(* CODESYS project HotWaterTank_student (2) (2).project

Project tree, tasks and I/O mapping:
  Device : CODESYS Control Win V3, 3S - Smart Software Solutions GmbH, version 3.5.17.10
    application Application
      libraries: Standard, * (System); Util, * (System)
      task MainTask (cyclic, interval t#10ms, priority 1) calls Model, PLC_PRG
      program Model [ST]: HeatingACT, SensorsACT, WaterLevelACT, OverpressureACT, InitializationACT
      visualisation Visualization
      program PLC_PRG [SFC]: Fill_active, Preheat_active_1, Operate_active, Init_Operate_active_active, Step0_Operate_active_active, Shutdown_active, HeatControl_active, Init_HeatControl_active_active, Step0_HeatControl_active_active, Empty_active, Fill_entry, Fill_exit, Preheat_entry, Preheat_exit, Operate_entry, Operate_exit, Shutdown_entry, Shutdown_exit, Empty_entry, Empty_exit
      trace Trace (task MainTask): Model.realTankLevel, Model.temperature
      global variables GVL
      function block GeneerinenSaato [ST]
      function block Heater [ST]
      function block SlowInlet [ST]
      function block FastInlet [ST]
      function block Heater2 [FBD]
      function block SlowInlet2 [FBD]
      function block FastInlet2 [FBD]
      visualisation Valvomo
  text list GlobalTextList
*)

// Device/Application/GVL
VAR_GLOBAL
	// Sensors:
	MinLevel:BOOL;
	LowLevel:BOOL;
	HighLevel:BOOL;
	MaxLevel:BOOL;
	MinTemp:BOOL;
	MaxTemp:BOOL;
	// Actuators:
	InletFast:BOOL;
	InletSlow:BOOL;
	Outlet:BOOL;
	Heat:BOOL;
END_VAR

// Device/Application/Model
PROGRAM Model
VAR
	// Define here the characteristics of the system.
	initialLevel :REAL := 0;		// Initial tank level, range [0..450], where 0=empty, 450=full tank.
	slowInlet :REAL := 10.0;		// Slow inlet flow rate in liters/s.
	fastInlet :REAL := 20.0;		// Fast inlet flow rate in liters/s.
	outlet	  :REAL := 15.0;		// Outlet flow rate in liters/s.
	posMinSensor	:REAL := 120;	// Position of min. sensor inside the tank. Range [0..450].
	posLowerSensor	:REAL := 170;	// Position of lower sensor inside the tank. Range [0..450].
	posUpperSensor	:REAL := 325;	// Position of upper sensor inside the tank. Range [0..450].
	posMaxSensor	:REAL := 375;	// Position of max sensor inside the tank. Range [0..450].
	minTemp   :REAL	:= 40.0;		// Minimum temperature sensor. Range [20..120].
	maxTemp   :REAL	:= 80.0;		// Maximum temperature sensor. Range [20..120].	
	heatCoeff :REAL := 3.0;			// Heating strenght of resistance.
	heatLooseCoeff	:REAL := 2.0;	// Cooling down coefficient of water.
END_VAR

VAR
	// Do not modify following variables unless you know what you are doing.
	initialized :BOOL := FALSE;
	tankLevel :REAL := 450.0;
	cycleTime :REAL := 10;			// PLC cycle time in ms. This should match the actual cycletime of the PLC.
	virtualTankLevel :REAL :=450;
	realTankLevel :REAL;
	slowValve :BOOL;
	fastValve :BOOL;
	outValve  :BOOL;
	heating   :BOOL;
	danger    :BOOL;
	overpress :REAL :=0.0;
	minSensor :BOOL;
	lowerSensor :BOOL;
	upperSensor :BOOL;
	maxSensor :BOOL;
	temperature :REAL :=20.0;
	minTempSensor :BOOL;
	maxTempSensor :BOOL;
	resistColor :DWORD := 16#00FF3A3A;
	resistBroken :BOOL;
	overheat :BOOL;
	tankExploded :BOOL;
	errorMsg :BOOL;
	blinkMsg :BLINK;
	startTrace :BOOL;
END_VAR

// Initialize system, only during reset.
IF NOT(initialized) THEN
	InitializationACT();
END_IF

// Read inputs from the controller's outputs:
IF NOT(tankExploded) THEN
	fastValve := GVL.InletFast;
	slowValve := GVL.InletSlow;
	outValve := GVL.Outlet;
	heating := GVL.Heat;
	startTrace := TRUE;
END_IF

// Determine the water level of tank based on inputs.
WaterLevelACT();

// Detect overpressure situations.
OverpressureACT();

// Run function taking care of the heating.
HeatingACT();

// Update sensors.
SensorsACT();

// Update model outputs / controller inputs:
GVL.MinLevel := minSensor;
GVL.LowLevel := lowerSensor;
GVL.HighLevel := upperSensor;
GVL.MaxLevel := maxSensor;
GVL.MinTemp := minTempSensor;
GVL.MaxTemp := maxTempSensor;

ACTION HeatingACT:
// Implementation of the heating
// Heating based on the level of the tank: the more water there is,
// the temperature will rise slower. Temperature refers to water temperature,
// not heating resistance.
IF heating AND (temperature < 100) AND (tankLevel < 449.9) AND NOT(resistBroken) THEN
	temperature := temperature + (heatCoeff*cycleTime/1000)*(tankLevel+50)/450.0;
END_IF

// If tank is empty, temperature drops to 0.
IF tankLevel > 449.9 THEN
	temperature := 20.0;
END_IF

// If heating is stopped or resistance is broken, temperature starts to drop.
IF (NOT(heating) OR resistBroken) AND temperature > 20.0 THEN
	temperature := temperature - heatLooseCoeff * cycleTime / 1000;
END_IF

// The following code takes care of the temperature resistance color
IF heating AND NOT(resistBroken) THEN
	IF resistColor < 16#FFFF3A3A AND NOT(overheat) THEN
		resistColor := resistColor + 16#01000000;
	END_IF
ELSE
	IF resistColor > 16#00FF3A3A AND NOT(overheat) THEN
		resistColor := resistColor - 16#01000000;	
	END_IF
END_IF

// If heating is turned on, but no water is in the tank, the resistance breaks
// once it reaches maximum value.
IF heating AND (tankLevel > 419.9) AND (resistColor >= 16#FFFF3A3A) THEN
	overheat := TRUE;
END_IF

IF heating AND overheat AND (tankLevel > 419.9) THEN
	resistColor := resistColor + 16#00000101;
END_IF
IF NOT(heating) AND overheat AND (resistColor > 16#FFFF3A3A) THEN
	resistColor := resistColor - 16#00000101;
END_IF
IF heating AND overheat AND (tankLevel < 419.9) AND (resistColor > 16#FFFF3A3A) THEN
	resistColor := resistColor - 16#00000101;
END_IF
IF NOT(heating) AND (resistColor <= 16#FFFF3A3A) THEN
	overheat := FALSE;
END_IF

IF heating AND (resistColor = 16#FFFFFFFF) AND (tankLevel > 419.9) THEN
	resistBroken := TRUE;
	resistColor := 16#00000000;
END_IF
END_ACTION

ACTION SensorsACT:
// Level sensors.
IF (tankLevel <= 450 - posMinSensor) THEN
	minSensor := TRUE;
ELSE
	minSensor := FALSE;
END_IF
IF (tankLevel <= 450 - posLowerSensor) THEN
	lowerSensor := TRUE;
ELSE
	lowerSensor := FALSE;
END_IF
IF (tankLevel <= 450 - posUpperSensor) THEN
	upperSensor := TRUE;
ELSE
	upperSensor := FALSE;
END_IF
IF (tankLevel <= 450 - posMaxSensor) THEN
	maxSensor := TRUE;
ELSE
	maxSensor := FALSE;
END_IF

// Temperature sensors.
IF temperature >= minTemp THEN
	minTempSensor := TRUE;
ELSE
	minTempSensor := FALSE;
END_IF

IF temperature >= maxTemp THEN
	maxTEmpSensor := TRUE;
ELSE
	maxTempSensor := FALSE;
END_IF
END_ACTION

ACTION WaterLevelACT:
// Implementation for the water level
// If slow inlet is TRUE, water level rises slow.
IF slowValve AND (virtualTankLevel > - 60) THEN
	virtualTankLevel := virtualTankLevel - slowInlet * cycleTime / 1000;
END_IF

// If fast inlet is TRUE, water level rises faster.
IF fastValve AND (virtualTankLevel > -60) THEN
	virtualTankLevel := virtualTankLevel - fastInlet * cycleTime / 1000;
END_IF

// Limits are set, so that "water" in the visualization does not go over or under the tank.
// Please note, that due to the visualization coordinates, 450 indicates an empty tank,
// while 0 indicates a full tank.
IF outValve THEN
	IF virtualTankLevel < 450.0 THEN
		virtualTankLevel := virtualTankLevel + outlet * cycleTime / 1000;
	ELSE
		virtualTankLevel := 450.0;
	END_IF
END_IF
IF (virtualTankLevel < 0.0) THEN
	tankLevel := 0.0;
ELSE
	tankLevel := virtualTankLevel;
END_IF

// Get real level of tank (0 means empty and 450 means full tank).
realTankLevel := 450.0 - tankLevel;
END_ACTION

ACTION OverpressureACT:
// Overpressure situation. A level below 0 indicates overpressure.
IF (virtualTankLevel < 0) THEN
	danger := TRUE;
	overpress := - virtualTankLevel * 0.6;
ELSE
	danger := FALSE;
END_IF

// If overpressure continues growing and it is not corrected, tank 
// "explodes" and error message is displayed.
IF overpress > 36.0 THEN
	tankExploded := TRUE;
	WHILE(1) DO
		// Infinite loop, need to cold restart for the system to work again.
		blinkMsg(ENABLE:=TRUE,TIMELOW:=T#1S,TIMEHIGH:=T#1S,OUT=>errorMsg);
	END_WHILE
END_IF
END_ACTION

ACTION InitializationACT:
tankLevel := 450.0 - initialLevel;
virtualTankLevel := 450.0 - initialLevel;

initialized := TRUE;
END_ACTION

END_PROGRAM

// Device/Application/SlowInlet
FUNCTION_BLOCK SlowInlet
VAR_INPUT
END_VAR
VAR_OUTPUT
	lock:BOOL;
END_VAR
VAR
END_VAR

IF(GVL.MaxLevel = TRUE) THEN
	GVL.InletSlow := FALSE;
	lock := TRUE;
END_IF

END_FUNCTION_BLOCK

// Device/Application/FastInlet
FUNCTION_BLOCK FastInlet
VAR_INPUT
END_VAR
VAR_OUTPUT
	lock:BOOL;
END_VAR
VAR
END_VAR

IF(GVL.MaxLevel = TRUE) THEN
	GVL.InletSlow := FALSE;
	lock := TRUE;
END_IF

END_FUNCTION_BLOCK

// Device/Application/PLC_PRG
PROGRAM PLC_PRG
VAR
	// You can declare here your variables:
	lampotila:GeneerinenSaato;
	pinta:GeneerinenSaato;
	heater:Heater2;
	nopee:FastInlet2;
	hidas:SlowInlet2;
	
	stopEmpty:BOOL := FALSE;
	
	InFill:BOOL;
	InPreheat:BOOL;
	InOperate:BOOL;
	InShutdown:BOOL;
	InEmpty:BOOL;
	
END_VAR

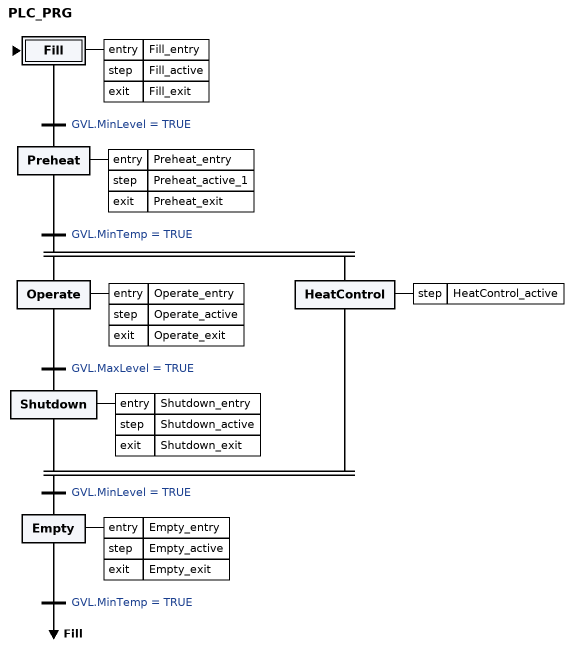
INITIAL_STEP Fill:
    Fill_entry(P1);  // entry action
    Fill_active(N);  // step action
    Fill_exit(P0);  // exit action
END_STEP
TRANSITION FROM Fill TO Preheat
    := GVL.MinLevel = TRUE;
END_TRANSITION
STEP Preheat:
    Preheat_entry(P1);  // entry action
    Preheat_active_1(N);  // step action
    Preheat_exit(P0);  // exit action
END_STEP
TRANSITION FROM Preheat TO (Operate, HeatControl)
    := GVL.MinTemp = TRUE;
END_TRANSITION
STEP Operate:
    Operate_entry(P1);  // entry action
    Operate_active(N);  // step action
    Operate_exit(P0);  // exit action
END_STEP
TRANSITION FROM Operate TO Shutdown
    := GVL.MaxLevel = TRUE;
END_TRANSITION
STEP Shutdown:
    Shutdown_entry(P1);  // entry action
    Shutdown_active(N);  // step action
    Shutdown_exit(P0);  // exit action
END_STEP
STEP HeatControl:
    HeatControl_active(N);  // step action
END_STEP
TRANSITION FROM (Shutdown, HeatControl) TO Empty
    := GVL.MinLevel = TRUE;
END_TRANSITION
STEP Empty:
    Empty_entry(P1);  // entry action
    Empty_active(N);  // step action
    Empty_exit(P0);  // exit action
END_STEP
TRANSITION FROM Empty TO Fill
    := GVL.MinTemp = TRUE;
END_TRANSITION

ACTION Fill_active:

Heat :=  FALSE;
IF (MinLevel = FALSE) THEN
	InletFast := TRUE;
	InletSlow := TRUE;
	Outlet := FALSE;
END_IF
END_ACTION

ACTION Preheat_active_1:
Heat := TRUE;
InLetSlow := TRUE;
InLetFast := FALSE;
pinta.high := GVL.LowLevel;
pinta.low := GVL.MinLevel;
GVL.Outlet := pinta.out;
pinta();
END_ACTION

ACTION Operate_active:
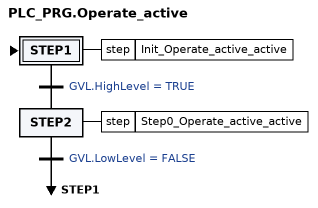
INITIAL_STEP STEP1:
    Init_Operate_active_active(N);  // step action
END_STEP
TRANSITION FROM STEP1 TO STEP2
    := GVL.HighLevel = TRUE;
END_TRANSITION
STEP STEP2:
    Step0_Operate_active_active(N);  // step action
END_STEP
TRANSITION FROM STEP2 TO STEP1
    := GVL.LowLevel = FALSE;
END_TRANSITION
END_ACTION

ACTION Init_Operate_active_active:

GVL.Outlet := FALSE;
GVL.InletFast := TRUE;
GVL.InletSlow := TRUE;
END_ACTION

ACTION Step0_Operate_active_active:

GVL.Outlet := TRUE;
GVL.InletFast := FALSE;
GVL.InletSlow := FALSE;
END_ACTION

ACTION Shutdown_active:
GVL.Outlet := TRUE;
GVL.InletFast := FALSE;
GVL.InletSlow := FALSE;
END_ACTION

ACTION HeatControl_active:
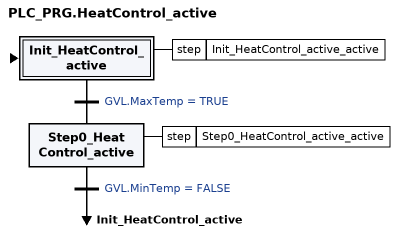
INITIAL_STEP Init_HeatControl_active:
    Init_HeatControl_active_active(N);  // step action
END_STEP
TRANSITION FROM Init_HeatControl_active TO Step0_HeatControl_active
    := GVL.MaxTemp = TRUE;
END_TRANSITION
STEP Step0_HeatControl_active:
    Step0_HeatControl_active_active(N);  // step action
END_STEP
TRANSITION FROM Step0_HeatControl_active TO Init_HeatControl_active
    := GVL.MinTemp = FALSE;
END_TRANSITION
END_ACTION

ACTION Init_HeatControl_active_active:
Heat := TRUE;
END_ACTION

ACTION Step0_HeatControl_active_active:
Heat := FAlSE;
END_ACTION

ACTION Empty_active:
Heat := FALSE;
GVL.InletFast := FALSE;
GVL.InletSlow := FALSE;
GVL.Outlet := TRUE;
END_ACTION

ACTION Fill_entry:
InFill := TRUE;
END_ACTION

ACTION Fill_exit:
InFill := FALSE;
END_ACTION

ACTION Preheat_entry:
InPreheat := TRUE;
END_ACTION

ACTION Preheat_exit:
InPreheat := FALSE;
END_ACTION

ACTION Operate_entry:
InOperate := TRUE;
END_ACTION

ACTION Operate_exit:
InOperate := False;
END_ACTION

ACTION Shutdown_entry:
InShutdown := TRUE;
END_ACTION

ACTION Shutdown_exit:
InShutdown := FALSE;
END_ACTION

ACTION Empty_entry:
InEmpty := TRUE;
END_ACTION

ACTION Empty_exit:
InEmpty := FALSE;
END_ACTION

END_PROGRAM

// Device/Application/GeneerinenSaato
FUNCTION_BLOCK GeneerinenSaato
VAR_INPUT
	high:BOOL;
	low:BOOL;
END_VAR
VAR_OUTPUT
	out:BOOL;
END_VAR
VAR
END_VAR

IF(high = TRUE) THEN
	out := TRUE;	
ELSIF (low = FALSE) THEN
	out := FALSE;
END_IF

END_FUNCTION_BLOCK

// Device/Application/Heater
FUNCTION_BLOCK Heater
VAR_INPUT
	in:BOOL;
END_VAR
VAR_OUTPUT
	lock:BOOL;
END_VAR
VAR
END_VAR

IF(GVL.MaxTemp = TRUE OR GVL.MinLevel = FALSE) THEN
	lock := TRUE;
	GVL.Heat := FALSE;
END_IF

END_FUNCTION_BLOCK

// Device/Application/Heater2
FUNCTION_BLOCK Heater2
VAR_INPUT
	in: BOOL;
END_VAR
VAR_OUTPUT
	lock: BOOL;
	out: BOOL;
END_VAR
VAR
END_VAR
VAR // added by the converter: edge detectors and wires of the graphical bodies
    _w1 : BOOL;
END_VAR

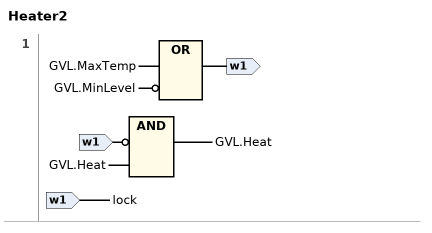
// NETWORK 1
_w1 := GVL.MaxTemp OR NOT GVL.MinLevel;
GVL.Heat := NOT _w1 AND GVL.Heat;
lock := _w1;

END_FUNCTION_BLOCK

// Device/Application/FastInlet2
FUNCTION_BLOCK FastInlet2
VAR_INPUT
	in:BOOL;
END_VAR
VAR_OUTPUT
	out:BOOL;
	lock:BOOL;
END_VAR
VAR
END_VAR

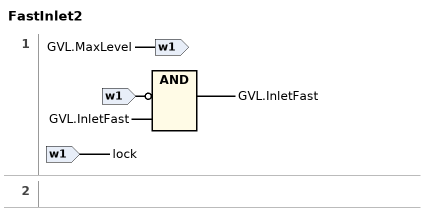
// NETWORK 1
GVL.InletFast := NOT GVL.MaxLevel AND GVL.InletFast;
lock := GVL.MaxLevel;

// NETWORK 2

END_FUNCTION_BLOCK

// Device/Application/SlowInlet2
FUNCTION_BLOCK SlowInlet2
VAR_INPUT
	in:BOOL;
END_VAR
VAR_OUTPUT
	lock:BOOL;
	out:BOOL;
END_VAR
VAR
END_VAR

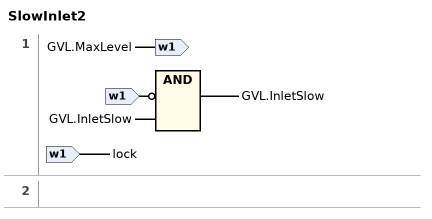
// NETWORK 1
GVL.InletSlow := NOT GVL.MaxLevel AND GVL.InletSlow;
lock := GVL.MaxLevel;

// NETWORK 2

END_FUNCTION_BLOCK

// Device/Application/Visualization
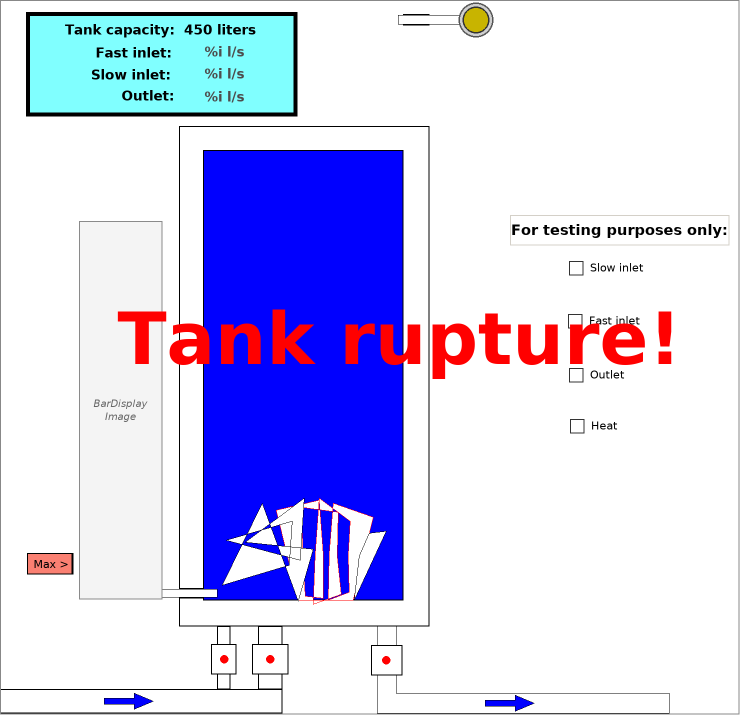
VISUALIZATION Visualization  // 740x715
    RoundedRectangle (179,126 250x500)
    Rectangle (203,150 200x450)
    Rectangle (203,150 200x450), tooltip "Current tank level"
        p2773130477: Model.tankLevel
    Checkbox (567,253 150x30), "Slow inlet", variable: GVL.InletSlow
    Checkbox (566,306 150x30), "Fast inlet", variable: GVL.InletFast
    Checkbox (567,360 150x30), "Outlet", variable: GVL.Outlet
    Checkbox (568,411 150x30), "Heat", variable: GVL.Heat
    Rectangle (217,626 13x63)
    Rectangle (0,689 282x24)
    Rectangle (258,626 24x63)
    RoundedRectangle (252,644 36x30)
    RoundedRectangle (211,644 25x30)
    Ellipse (266,655 8x8)
    Ellipse (220,655 8x8)
    Ellipse (266,655 8x8), invisible if: NOT(Model.fastValve)
    Ellipse (220,655 8x8), invisible if: NOT(Model.slowValve)
    Polygon (377,626) (377,713) (669,713) (669,693) (396,693) (396,626)
    RoundedRectangle (371,645 31x30)
    Ellipse (382,656 8x8)
    Ellipse (382,656 8x8), invisible if: NOT(Model.outValve)
    Meter360 (473,34 157x148), value: Model.overpress, style: Meter-Meter360-Gray, scale format: %.1f, scale 0..40
        p518627256: Gauge
    Rectangle (455,11 200x192), invisible if: Model.danger
    Group (398,0 98x40), tooltip "Max. sensor."
        p2738717112: (580 - Model.posMaxSensor)
        Rectangle (5,14 26x11)
        Polygon (89,15) (0,15) (0,19) (0,24) (89,24)
        Lamp1 (58,0 40x40), tooltip "Max. sensor", variable: Model.maxSensor, style: Lamp-Lamp1-Yellow
    Group (398,0 98x40), tooltip "Upper sensor."
        p2738717112: (580 - Model.posUpperSensor)
        Rectangle (5,14 26x11)
        Polygon (89,15) (0,15) (0,20) (0,24) (89,24)
        Lamp1 (58,0 40x40), tooltip "Upper sensor", variable: Model.upperSensor, style: Lamp-Lamp1-Yellow
    Group (398,0 98x40), tooltip "Min. sensor."
        p2738717112: (580 - Model.posMinSensor)
        Rectangle (5,14 26x11)
        Polygon (89,15) (0,15) (0,20) (0,24) (89,24)
        Lamp1 (58,0 40x40), tooltip "Min sensor", variable: Model.minSensor, style: Lamp-Lamp1-Yellow
    Group (398,0 98x40), tooltip "Lower sensor."
        p2738717112: (580 - Model.posLowerSensor)
        Rectangle (5,14 26x11)
        Polygon (89,15) (0,15) (0,20) (0,24) (89,24)
        Lamp1 (58,0 40x40), tooltip "Lower sensor", variable: Model.lowerSensor, style: Lamp-Lamp1-Yellow
    Polygon (485,700) (485,706) (515,706) (515,711) (534,703) (515,695) (515,700), invisible if: NOT(Model.outValve)
    Polygon (104,698) (104,704) (134,704) (134,709) (153,701) (134,693) (134,698), invisible if: NOT(Model.slowValve OR Model.fastValve)
    Polygon (298,600) (276,510) (319,500) (323,554) (323,598) (305,596) (303,557) (301,507) (338,512) (337,556) (341,594) (313,604) (315,554) (319,498) (350,521) (348,555) (349,592) (328,600) (329,554) (333,503) (373,517) (353,600) (353,600), invisible if: Model.resistBroken
    Polygon (298,600) (276,510) (319,500) (323,554) (323,598) (305,596) (303,557) (301,507) (338,512) (337,556) (341,594) (313,604) (315,554) (319,498) (350,521) (348,555) (349,592) (328,600) (329,554) (333,503) (373,517) (353,600) (353,600), invisible if: Model.resistBroken
        p3450524324: Model.resistColor
    Group (31,549 42x31)
        p2738717112: -(Model.minTemp-20)/100*308
        RoundedRectangle (0,4 42x21), colour toggle: Model.minTempSensor
        Label (2,0 40x31), "Min >"
    Group (27,542 46x45)
        p2738717112: -(Model.maxTemp-20)/100*308
        RoundedRectangle (0,11 45x21), colour toggle: Model.maxTempSensor
        Label (2,0 44x45), "Max >"
    Rectangle (179,588 24x10)
    Polygon (217,589) (127,589) (127,597) (217,597) (217,593)
    BarDisplayImage (79,221 83x378), value: Model.temperature, style: BarDisplayImage-Gray, scale format: %.1f, scale 20..120
        p518627256: °C
    Textfield (61,249 677x179), "Tank rupture!", invisible if: NOT(Model.errorMsg)
    Polygon (298,601) (262,503) (222,585) (289,565) (292,521) (226,540) (300,560) (304,498) (245,542) (313,549), invisible if: NOT(Model.resistBroken)
    Polygon (354,600) (359,556) (369,533) (386,531), invisible if: NOT(Model.resistBroken)
    Textfield (510,215 219x30), "For testing purposes only:"
    Rectangle (26,12 271x104)
    Label (39,13 243x34), "Tank capacity: 450 liters"
    Label (74,36 120x34), "Fast inlet:"
    Label (69,58 124x34), "Slow inlet:"
    Label (86,79 124x34), "Outlet:"
    Textfield (180,37 89x30), "%i l/s", text variable: Model.fastInlet
    Textfield (180,59 89x30), "%i l/s", text variable: Model.slowInlet
    Textfield (180,82 89x30), "%i l/s", text variable: Model.outlet
END_VISUALIZATION

// Device/Application/Valvomo
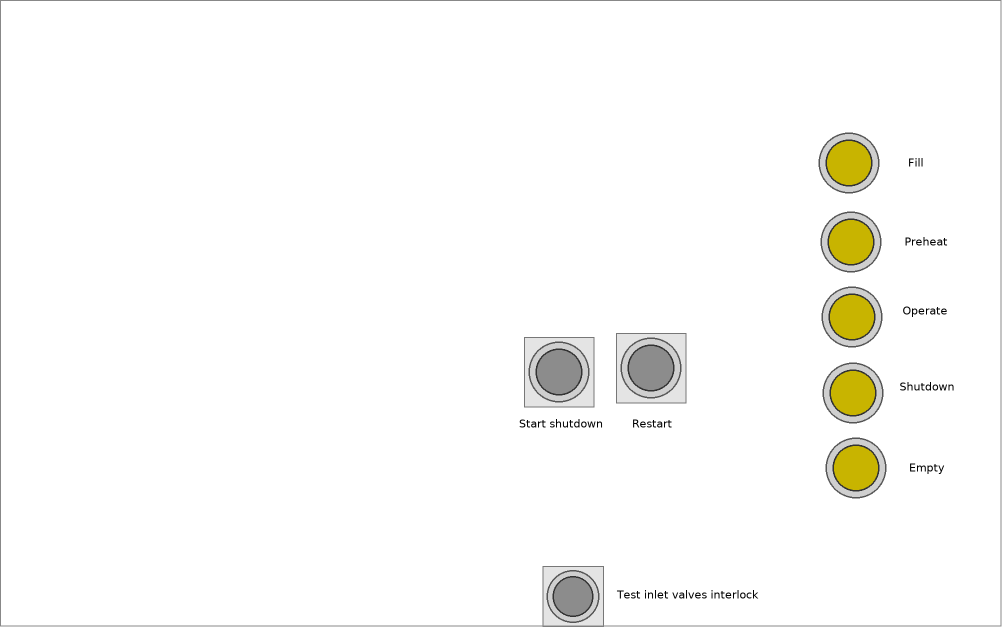
VISUALIZATION Valvomo  // 1002x627
    Lamp1 (817,282 70x70), variable: PLC_PRG.InOperate, style: Lamp-Lamp1-Yellow
    Lamp1 (818,358 70x70), variable: PLC_PRG.InShutdown, style: Lamp-Lamp1-Yellow
    Lamp1 (821,433 70x70), variable: PLC_PRG.InEmpty, style: Lamp-Lamp1-Yellow
    Lamp1 (816,207 70x70), variable: PLC_PRG.InPreheat, style: Lamp-Lamp1-Yellow
    Lamp1 (814,128 70x70), variable: PLC_PRG.InFill, style: Lamp-Lamp1-Yellow
    PushSwitch (524,337 70x70), behaviour: TOGGLE, style: Switch-PushSwitch-Gray
    PushSwitch (616,333 70x70), behaviour: TOGGLE, style: Switch-PushSwitch-Gray
    PushSwitch (541,566 64x61), behaviour: TOGGLE, style: Switch-PushSwitch-Gray
    Label (486,409 150x30), "Start shutdown"
    Label (577,409 150x30), "Restart"
    Label (613,580 150x30), "Test inlet valves interlock"
    Label (852,453 150x30), "Empty"
    Label (852,372 150x30), "Shutdown"
    Label (850,296 150x30), "Operate"
    Label (851,227 150x30), "Preheat"
    Label (841,148 150x30), "Fill"
END_VISUALIZATION
